{attribute 'qualified_only'}
{attribute 'strict'}
TYPE E_MOTOR_COMMAND :
(
	NONE	:= 0,
	
	// Commands corresponding to events - MUST match E_MOTOR_EVENT !!!
	RESET,
	INIT,
	STOP,
	ENABLE,
	DISABLE,
	MOTOR_MOVE,
	SET_POSITION,
	CLEAR_NOVRAM
);
END_TYPE

(* stored: Version 1.1.0.1, ProductVersion 3.1.4022.16
   DUT E_MOTOR_COMMAND: Id {384c1f9b-10c2-4511-9e8a-004d22171a66} *)
